FUNCTION_BLOCK PUBLIC PAPoint EXTENDS ACObject IMPLEMENTS IACPoint
VAR_INPUT
END_VAR
VAR_OUTPUT
END_VAR
VAR
	_PAEdges : ARRAY [1..GCL.cEdgeMAX] OF IACEdge;
	_Parent : IACComponent;	
END_VAR

METHOD AddEdge : BOOL
VAR_INPUT
	edge : IACEdge;
END_VAR
VAR
	i: INT;
END_VAR
IF edge = 0 THEN
	AddEdge := FALSE;
	RETURN;
END_IF

// 1. Check if edge already exists in the array because of online change
FOR i:=1 TO GCL.cEdgeMAX BY 1
  DO
    IF _PAEdges[i] <> 0 THEN
		IF _PAEdges[i] = edge THEN
			AddEdge := FALSE;
			RETURN;						
		END_IF
		(*IF _PAEdges[i].Compare(edge) THEN
			AddEdge := FALSE;
			RETURN;						
		END_IF*)
	ELSE
		EXIT;
	END_IF
END_FOR;
// 2. If the child doesn't exist, add to _Childs-List
FOR i:=1 TO GCL.cEdgeMAX BY 1
  DO
    IF _PAEdges[i] = 0 THEN
		AddEdge := TRUE;
		_PAEdges[i] := edge;
		EXIT;
	END_IF
END_FOR;
END_METHOD

PROPERTY ConnectionList : ARRAY [1..GCL.cEdgeMAX] OF IACEdge
GET
ConnectionList := _PAEdges;
END_GET
END_PROPERTY

METHOD FB_init : BOOL
VAR_INPUT
	bInitRetains : BOOL; // if TRUE, the retain variables are initialized (warm start / cold start)
	bInCopyCode : BOOL;  // if TRUE, the instance afterwards gets moved into the copy code (online change)
	parent : IACComponent;
END_VAR

VAR
	isValidRef: BOOL;
END_VAR
IF parent <> 0 THEN
	_Parent := parent;
END_IF
IncFBInitCount();
END_METHOD

METHOD PUBLIC FB_postinit
VAR_INPUT
		root : IACVariobatch;
END_VAR
VAR
	i: INT;
	thisPoint : IACPoint;
	iPoint : IACPoint;
END_VAR
SUPER^.FB_postinit(root);
thisPoint := THIS^;
FOR i:=1 TO GCL.cEdgeMAX BY 1
  DO
    IF _PAEdges[i] <> 0 THEN
		iPoint := _PAEdges[i].Source;
		IF iPoint = thisPoint THEN
			_PAEdges[i].FB_postinit(root);			
		END_IF
	ELSE
		EXIT;
	END_IF
END_FOR;
END_METHOD

METHOD FindObjectInChilds : IACObject
VAR_INPUT
	instanceID	: UDINT;
END_VAR
VAR
	i: INT;
	currentEdge : IACEdge;	
END_VAR
FOR i:=1 TO GCL.cEdgeMAX BY 1
  DO
    IF _PAEdges[i] <> 0 THEN
		currentEdge := _PAEdges[i];
		IF currentEdge.InstanceID = instanceID THEN
			FindObjectInChilds := currentEdge;
			RETURN;
		END_IF
	ELSE
		EXIT;
	END_IF
END_FOR;
FindObjectInChilds := 0;
END_METHOD

METHOD PUBLIC GetAllocatedEdge : IACEdge
VAR_INPUT
	paFunction : IPAProcessFunction;
END_VAR
VAR
	i: INT;
END_VAR
//IPAProcessFunction
IF paFunction = 0 THEN
	GetAllocatedEdge := 0;
	RETURN;
END_IF
// 1. Check if edge already exists in the array because of online change
FOR i:=1 TO GCL.cEdgeMAX BY 1
  DO
    IF _PAEdges[i] <> 0 THEN
		IF _PAEdges[i].AllocatedByFunction = 0 THEN
			GetAllocatedEdge := 0;
			RETURN;
		END_IF
		IF _PAEdges[i].AllocatedByFunction = paFunction THEN
			GetAllocatedEdge := _PAEdges[i];
			RETURN;			
		END_IF
	ELSE
		EXIT;
	END_IF
END_FOR;
GetAllocatedEdge := 0;
END_METHOD

PROPERTY Parent : IACComponent
GET
Parent := _Parent;
END_GET
END_PROPERTY

PROPERTY TypeOfACObject : TypeOfACObjectEnum
GET
TypeOfACObject := TypeOfACObjectEnum.Point;
END_GET
END_PROPERTY

END_FUNCTION_BLOCK

(* stored: Version 1.1.0.1, ProductVersion 3.1.4022.7
   POU PAPoint: Id {cf190ec0-0be4-41a4-be77-f8eeefca0242}, SpecialFunc None
   Method AddEdge: Id {02f5fa6b-3258-4ee4-94c5-89972ed0c28f}
   Property ConnectionList: Id {514c623b-23da-442d-98fb-3b1f89528ee9}
   Get Get: Id {87203c66-6133-4bcf-b4ef-4775346c2995}
   Method FB_init: Id {786d5e53-ad5c-4778-9604-f0ca0b25d3d9}
   Method FB_postinit: Id {b846993c-3769-4e27-8453-066b1c284f57}
   Method FindObjectInChilds: Id {002a08a5-09ff-4cdb-b62c-71ddb81c35a1}
   Method GetAllocatedEdge: Id {5ae7f375-98ad-4a6e-a43d-d860347cc161}
   Property Parent: Id {73fa2ae6-20b3-4e9d-9852-bb2cdb3252bb}
   Get Get: Id {f9de2fbd-ebec-46eb-9843-07dc977bc203}
   Property TypeOfACObject: Id {8289de43-5b68-4d46-8afd-1c39b6fcb123}
   Get Get: Id {f37f76d0-fdd8-4831-baa3-b7f2c307c423} *)
